// Mitsubishi GX Works2 project: 인터락구현   PLC: Q02/Q02H

PROGRAM MAIN
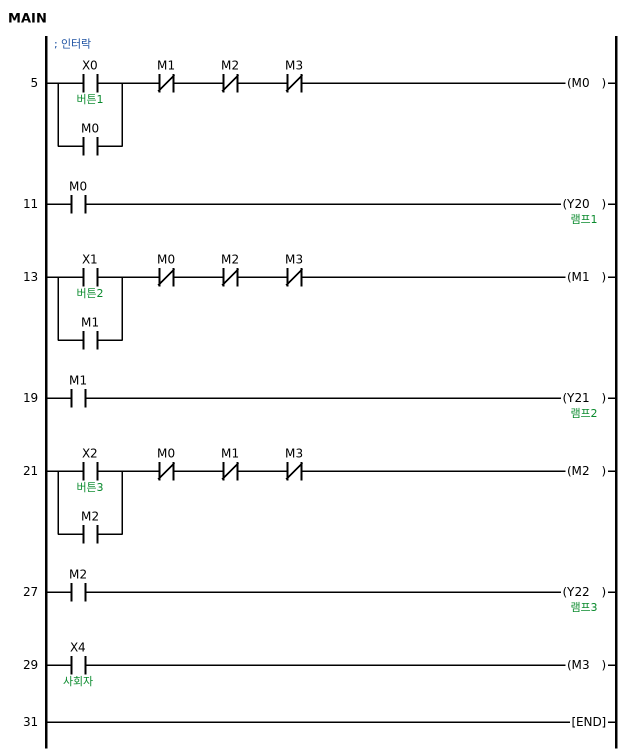
; 인터락
5     LD      X0  ; 버튼1
      OR      M0
      ANI     M1
      ANI     M2
      ANI     M3
      OUT     M0
11    LD      M0
      OUT     Y20  ; 램프1
13    LD      X1  ; 버튼2
      OR      M1
      ANI     M0
      ANI     M2
      ANI     M3
      OUT     M1
19    LD      M1
      OUT     Y21  ; 램프2
21    LD      X2  ; 버튼3
      OR      M2
      ANI     M0
      ANI     M1
      ANI     M3
      OUT     M2
27    LD      M2
      OUT     Y22  ; 램프3
29    LD      X4  ; 사회자
      OUT     M3
31    END
END_PROGRAM

// device comments not shown above
M4  ; 3
